TYPE DUT_HMI_06_MANUALS :
STRUCT
	PS : ARRAY[0..CNC.NUM_MAX_MANUALS_06-1] OF BOOL;
	LS : ARRAY[0..CNC.NUM_MAX_MANUALS_06-1] OF BOOL;
END_STRUCT
END_TYPE

(* stored: Version 1.1.0.1, ProductVersion 3.1.4024.13
   DUT DUT_HMI_06_MANUALS: Id {eee1e142-48ad-418e-a713-172e101d8292} *)
